FUNCTION_BLOCK Test_AggregateResult_Aborted EXTENDS T_UnitTestBase
VAR
    ResultAggregate : T_ResultAggregate;
    Execution1      : T_Execution;
    Execution2      : T_Execution;
    Execution3      : T_Execution;
END_VAR

{attribute 'analysis' := '-33'} // inhibit unused variable warning
METHOD RunTest
IF Retest THEN
    SUPER^.Init();
END_IF

IF TestCompleted THEN
    RETURN;
END_IF

F_Inc(CycleCount);
IF CycleCount > 1000 THEN
    Fail(Message := 'Timeout');
END_IF

ResultAggregate.Clear();

ResultAggregate.AddResult(Execution1);
ResultAggregate.AddResult(Execution2);
ResultAggregate.AddResult(Execution3);

AssertIsTrue(Condition := ResultAggregate.Aborted = FALSE,
             Message   := 'ResultAggregate.Aborted is not false');

Execution1.Start();
Execution1.SetBusy();
Execution1.Abort();
Execution1.SetAborted();

Execution2.Start();
Execution2.SetBusy();
Execution2.Abort();
Execution2.SetAborted();

Execution3.Start();
Execution3.SetBusy();
Execution3.Abort();
Execution3.SetAborted();

AssertIsTrue(Condition := ResultAggregate.Aborted,
             Message   := 'ResultAggregate.Aborting is false');

TestCompleted := TRUE;
END_METHOD

END_FUNCTION_BLOCK

(* stored: Version 1.1.0.1, ProductVersion 3.1.4024.15
   POU Test_AggregateResult_Aborted: Id {4a1005d9-5a4e-41b6-b8ab-e43407083448}, SpecialFunc None
   Method RunTest: Id {2d34d322-da1b-484f-817c-82e5d6e016a3} *)
